TYPE User :
STRUCT
	{attribute 'TcEncoding':='UTF-8'}
	Email: STRING;
	{attribute 'TcEncoding':='UTF-8'}
	Password: STRING(30);
	{attribute 'TcEncoding':='UTF-8'}
	Name: STRING;
	{attribute 'TcEncoding':='UTF-8'}
	Phone: STRING(20);
	Permissions: Permissions;
END_STRUCT
END_TYPE

(* stored: Version 1.1.0.1, ProductVersion 3.1.4024.4
   DUT User: Id {34c6725e-4b54-439e-9ba3-c63eef7afe35} *)
